PROGRAM MAIN
VAR
	fbConveyorSystem 		: FB_ConveyorSystem();
	sState 					: STRING;
	nCount 					: INT;
	bPressEmergencyStop 	: BOOL;
	bPressStart 			: BOOL;
	bPressStop 				: BOOL;
	bDetectedPartSensor1 	: BOOL;
	bDetectedWeightSensor 	: BOOL;
	bDetectedPartSensor2 	: BOOL;
END_VAR

fbConveyorSystem(bPressEmergencyStop := bPressEmergencyStop,
				 bPressStart := bPressStart,
				 bPressStop := bPressStop,
				 bDetectedPartSensor1 := bDetectedPartSensor1,
				 bDetectedWeightSensor := bDetectedWeightSensor,
				 bDetectedPartSensor2 := bDetectedPartSensor2);
				 
sState := fbConveyorSystem.ipState.Description;
nCount := fbConveyorSystem.nCount;

bPressEmergencyStop := FALSE;
bPressStart := FALSE;
bPressStop := FALSE;

END_PROGRAM

(* stored: Version 1.1.0.1, ProductVersion 3.1.4024.12
   POU MAIN: Id {2ac301fe-ca5a-4f78-8ed4-0564a60cfe4d}, SpecialFunc None *)
